// TIA Portal V18 export
// export: Created 2026-03-12T16:04:35.5063979Z, ExportSetting WithDefaults, DisplayName Totally Integrated Automation Portal, DisplayVersion V18 Update 5, DisplayName TIA Portal Openness, DisplayVersion V18 Update 5, DisplayName TIA Portal Version Control Interface, DisplayVersion V18, DisplayName SINAMICS Startdrive Advanced, DisplayVersion V18, DisplayName SINAMICS Startdrive G130, G150, S120, S150, SINAMICS MV, S210, DisplayVersion V18, DisplayName SINAMICS Startdrive G110M, G120, G120C, G120D, G120P, G115D, DisplayVersion V18, DisplayName STEP 7 Professional, DisplayVersion V18 Update 5, DisplayName STEP 7 Safety, DisplayVersion V18, DisplayName WinCC Professional, DisplayVersion V18 Update 5
FUNCTION_BLOCK "FB MODBUS SCAN DRIVERS"   // FB19, LAD
TITLE = Function Block MODBUS SCAN DRIVERS: Varredura de drivers
{ S7_Optimized_Access := 'TRUE' }
VERSION : 0.1
// stored: AutoNumber true, IsIECCheckEnabled false, IsRetainMemResEnabled false, MemoryReserve 100, SetENOAutomatically false, UDAEnableTagReadback false
   VAR_INPUT
      IS_MMW : Bool;
      DONE : Bool;
      ERROR : Bool;
      QTD_DRIVER : Int;
      ID_START_DRIVER : Int;
      "TAG_N°_DRIVER" : Int;
      "TAG_N°_MMW" : Int;
      UPDATE_TIME : Time;
   END_VAR
   VAR_OUTPUT
      MODBUS_ID : Int;
      INDEX_ADDR : Int;
      INDEX_DRIVER : Int;
      TRIGGER : Bool;
   END_VAR
   VAR
      CHANGE_DRIVER : Bool;
      AUX_CHANGE : Bool;
      AUX_FINISH : Bool;
      AUX1 : Bool;
      AUX2 : Bool;
      AUX3 : Bool;
      TAGS : Int := 3;
      "TIMER" : IEC_TIMER;
      TIMER_2 { S7_SetPoint := 'True'} : IEC_TIMER;
   END_VAR
   VAR_TEMP   // added for the SCL form of the ladder/FBD networks
      _w1 : Bool;
      _w2 : Bool;
      _w3 : Bool;
      _w4 : Bool;
      _w5 : Bool;
      _w6 : Bool;
   END_VAR
BEGIN

REGION Network 1: Geração de variáveis para controle da varredura em "malha fechada"
   // Controle de malha fechado do Bloco modbus_Master.
   // O mesmo só pode ser chamado uma vez por módulo, ou seja necessita que seja multiplexado para atender mais de um escravo.
   // Para a lógica é usado um contato TOF, para controle do intervelo de tempo em que deve ser agregado o valor no INDEX(indice).
   // Após o telegrama ser encaminhado, sendo ele "True" ou "False" para DONE. O mesmo irá realimentar a malha de controle para que o próximo escravo seja chamado.
   // A situação acontece de igual forma para ERROR.
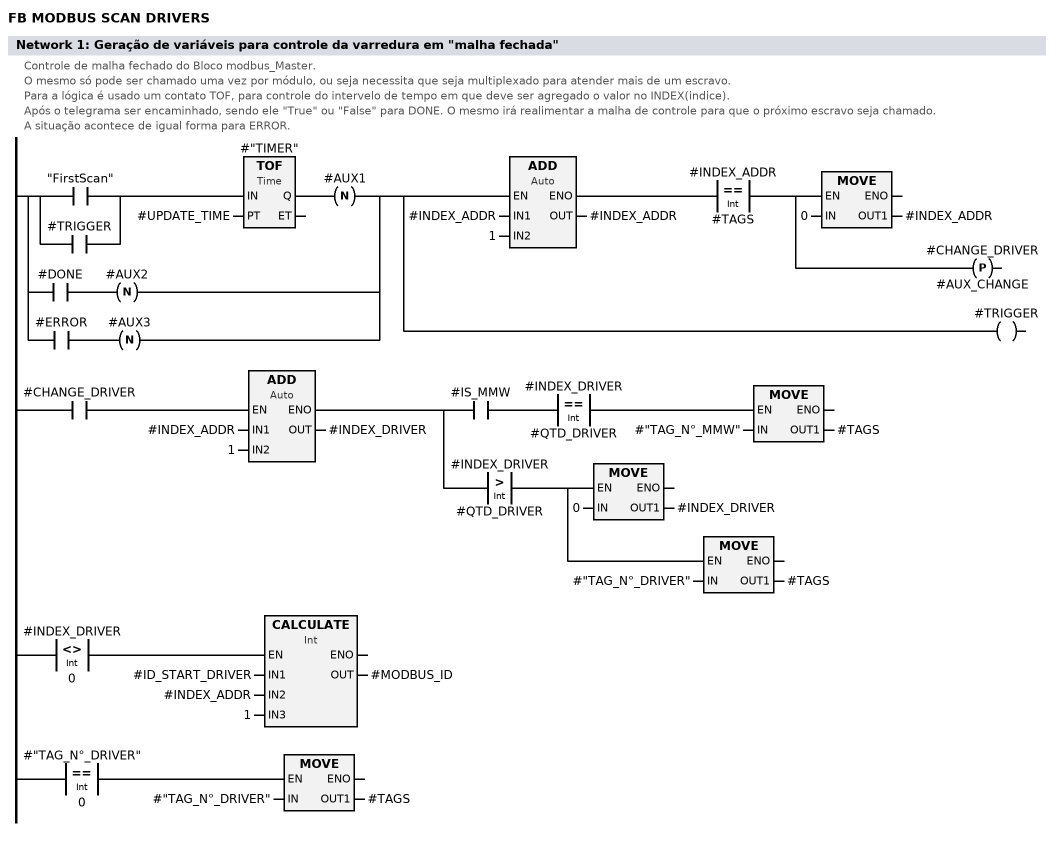
   #"TIMER".TOF(IN := "FirstScan" OR #TRIGGER, PT := #UPDATE_TIME);
   #_w1 := NOT #"TIMER".Q AND #AUX1;   // falling edge
   #AUX1 := #"TIMER".Q;
   #_w2 := NOT #DONE AND #AUX2;   // falling edge
   #AUX2 := #DONE;
   #_w3 := NOT #ERROR AND #AUX3;   // falling edge
   #AUX3 := #ERROR;
   #_w4 := #_w1 OR #_w2 OR #_w3;
   IF #_w4 THEN #INDEX_ADDR := #INDEX_ADDR + 1; END_IF;
   #_w5 := #_w4 AND (#INDEX_ADDR = #TAGS);
   IF #_w5 THEN #INDEX_ADDR := 0; END_IF;
   #CHANGE_DRIVER := #_w5 AND NOT #AUX_CHANGE;   // rising edge
   #AUX_CHANGE := #_w5;
   #TRIGGER := #_w4;
   IF #CHANGE_DRIVER THEN #INDEX_DRIVER := #INDEX_ADDR + 1; END_IF;
   IF #CHANGE_DRIVER AND #IS_MMW AND (#INDEX_DRIVER = #QTD_DRIVER) THEN #TAGS := #"TAG_N°_MMW"; END_IF;
   #_w6 := #CHANGE_DRIVER AND (#INDEX_DRIVER > #QTD_DRIVER);
   IF #_w6 THEN
       #INDEX_DRIVER := 0;
       #TAGS := #"TAG_N°_DRIVER";
   END_IF;
   IF #INDEX_DRIVER <> 0 THEN #MODBUS_ID := #ID_START_DRIVER + #INDEX_ADDR - 1; END_IF;
   IF #"TAG_N°_DRIVER" = 0 THEN #TAGS := #"TAG_N°_DRIVER"; END_IF;
END_REGION
END_FUNCTION_BLOCK
